Omron CX-Programmer project NewProject (CX-Programmer 9.61)

# PLC conveyor_1: CP1E E20

## Global symbols (name address type ; comment)
0.00 BOOL  ; START
0.01 BOOL  ; E-STOP
0.02 BOOL  ; SENSOR 1
0.03 BOOL  ; SENSOR 2
0.04 BOOL  ; STOP
100.00 BOOL  ; CONVEYOR 2
100.01 BOOL  ; CONVEYOR  1
100.02 BOOL  ; MAGAZINE
100.03 BOOL  ; SILINDER 1
100.04 BOOL  ; INDIKATOR SENSOR 1
100.05 BOOL  ; SILINDER 2
100.06 BOOL  ; INDIKATOR SENSOR 2

## Program NewProgram1 (cyclic task 0)

### Section Section1

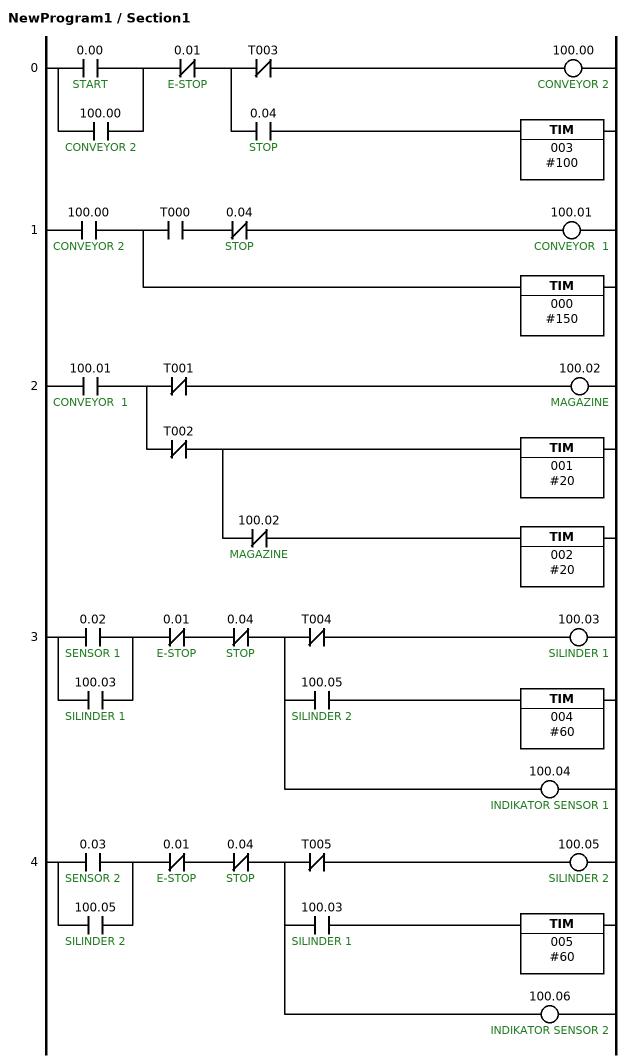
; rung 0
LD 0.00  ; START
OR 100.00  ; CONVEYOR 2
ANDNOT 0.01  ; E-STOP
OUT TR0
ANDNOT T003
OUT 100.00  ; CONVEYOR 2
LD TR0
AND 0.04  ; STOP
TIM 003 #100
; rung 1
LD 100.00  ; CONVEYOR 2
OUT TR0
AND T000
ANDNOT 0.04  ; STOP
OUT 100.01  ; CONVEYOR  1
LD TR0
TIM 000 #150
; rung 2
LD 100.01  ; CONVEYOR  1
OUT TR0
ANDNOT T001
OUT 100.02  ; MAGAZINE
LD TR0
ANDNOT T002
TIM 001 #20
ANDNOT 100.02  ; MAGAZINE
TIM 002 #20
; rung 3
LD 0.02  ; SENSOR 1
OR 100.03  ; SILINDER 1
ANDNOT 0.01  ; E-STOP
ANDNOT 0.04  ; STOP
OUT TR0
ANDNOT T004
OUT 100.03  ; SILINDER 1
LD TR0
AND 100.05  ; SILINDER 2
TIM 004 #60
LD TR0
OUT 100.04  ; INDIKATOR SENSOR 1
; rung 4
LD 0.03  ; SENSOR 2
OR 100.05  ; SILINDER 2
ANDNOT 0.01  ; E-STOP
ANDNOT 0.04  ; STOP
OUT TR0
ANDNOT T005
OUT 100.05  ; SILINDER 2
LD TR0
AND 100.03  ; SILINDER 1
TIM 005 #60
LD TR0
OUT 100.06  ; INDIKATOR SENSOR 2

### Section END
; rung 0
END(001)